// TIA Portal V17 export
// export: Created 2026-04-13T11:12:04.3028038Z, ExportSetting WithDefaults, DisplayName Totally Integrated Automation Portal, DisplayVersion V17 Update 4, DisplayName TIA Portal Openness, DisplayVersion V17 Update 4, DisplayName TIA Portal Version Control Interface, DisplayVersion V17, DisplayName SINAMICS Startdrive Advanced, DisplayVersion V17, DisplayName SINAMICS Startdrive G130, G150, S120, S150, SINAMICS MV, S210, DisplayVersion V17, DisplayName SINAMICS Startdrive G110M, G120, G120C, G120D, G120P, G115D, DisplayVersion V17, DisplayName STEP 7 Professional, DisplayVersion V17 Update 4, DisplayName STEP 7 Safety, DisplayVersion V17, DisplayName WinCC Professional, DisplayVersion V17 Update 4
DATA_BLOCK "BY1"   // DB9
{ S7_Optimized_Access := 'TRUE' }
VERSION : 0.1
// stored: AutoNumber true, DBAccessibleFromOPCUA true, DBAccessibleFromWebserver true, IsOnlyStoredInLoadMemory false, IsRetainMemResEnabled false, IsWriteProtectedInAS false, MemoryReserve 100
   VAR
      MBY等待保压 : Bool := FALSE;
      MBY正在充气 : Bool := TRUE;
      MBY保压不佳 : Bool := FALSE;
      MBY正在保压 : Bool := FALSE;
      MBY保压正常 : Bool := FALSE;
      MBY保压 : Bool := TRUE;
      MQT其他阀 : Bool := FALSE;
      MCQ充气阀 : Bool := FALSE;
      当前阶段 : Int := 1;
   END_VAR
   VAR RETAIN
      SV低设定 : Real := 1000.0;
      SV高设定 : Real := 3000.0;
      SV保压差值 : Real := 1000.0;
      SV保压时 : UInt := 0;
      SV保压分 : UInt := 0;
      SV保压秒 : UInt := 30;
   END_VAR
   VAR
      PV塔内压力 : Real := 0.0;
      PV保压前 : Real := 1016.367;
      PV保压后 : Real := 1016.367;
      PV当前差值 : Real := 0.0;
      PV保压时 : UInt := 0;
      PV保压分 : UInt := 0;
      PV保压秒 : UInt := 30;
      BY保压重置 : Bool := FALSE;
   END_VAR
BEGIN
END_DATA_BLOCK
